(* CoDeSys 2.3 export: GVL_APBOOL.EXP *)

(* Global variable list: GVL_APBool *)
VAR_GLOBAL CONSTANT
    WarmWait :BYTE:=0;    (*отложенный старт*)
    DynContr :BYTE:=1;    (*динамическое управление*)
    RotOn    :BYTE:=2;    (*качание*)
END_VAR
